FUNCTION FC10_Relaisschakel : BOOL
VAR_INPUT
	relaisNr : BOOL;
END_VAR
VAR
END_VAR

// NETWORK 1

END_FUNCTION

(* stored: Version 1.1.0.1, ProductVersion 3.1.4024.12
   POU FC10_Relaisschakel: Id {7dd28e65-b99d-40d7-b063-bf3b55816f4c}, SpecialFunc None *)
